PROGRAM PRG_MotorDrive
VAR
	fbEnableAxes: FB_EnableAxes;
	fbHalt1: MC_Halt;
	fbMoveVelocityFw: MC_MoveVelocity;
	fbMoveVelocityBw: MC_MoveVelocity;
	fbTON1: TON;
	fbRTrigMoveFw: R_TRIG;
	fbRTrigMoveBw: R_TRIG;
	fbRTrigHalt: R_TRIG;
	nAutoState: INT;
	nSpeed: INT := 400; //degrees/sec
END_VAR

fbEnableAxes.bEnableAxes := TRUE;
fbRTrigMoveFW(CLK:=GVL.bButtonFw, Q=>);
fbRTrigMoveBW(CLK:=GVL.bButtonBw, Q=>);
fbRTrigHalt(CLK:=GVL.bButtonHalt, Q=>);

IF fbRTrigMoveFw.Q THEN
	fbHalt1.Execute := FALSE;
	fbMoveVelocityBw.Execute := FALSE;
	fbMoveVelocityFw.Execute := TRUE;
END_IF

IF fbRTrigMoveBw.Q THEN
	fbHalt1.Execute := FALSE;
	fbMoveVelocityFw.Execute := FALSE;
	fbMoveVelocityBw.Execute := TRUE;
END_IF

IF fbRTrigHalt.Q THEN
	fbHalt1.Execute := TRUE;
	fbMoveVelocityFw.Execute := FALSE;
	fbMoveVelocityBw.Execute := FALSE;
END_IF

IF GVL.bButtonAuto THEN
	CASE nAutoState OF
		0: //Initialize auto motion
			fbHalt1.Execute := FALSE;
			fbMoveVelocityFw.Execute := FALSE;
			fbMoveVelocityBw.Execute := FALSE;
			nAutoState := 1;
		1: //Move forward
			fbTON1(IN:=TRUE, PT:=T#4S, Q=>, ET=>);
			fbMoveVelocityFw.Execute := TRUE;
			IF fbTON1.Q THEN
				fbTON1(IN:=FALSE);
				nAutoState := 2;	
			END_IF
		2: //Halt
			fbTON1(IN:=TRUE, PT:=T#2S, Q=>, ET=>);
			fbMoveVelocityFw.Execute := FALSE;
			fbHalt1.Execute := TRUE;
			IF fbTON1.Q THEN
				fbTON1(IN:=FALSE);
				nAutoState := 3;	
			END_IF
		3: //Move backward
			fbTON1(IN:=TRUE, PT:=T#4S, Q=>, ET=>);
			fbHalt1.Execute := FALSE;
			fbMoveVelocityBw.Execute := TRUE;
			IF fbTON1.Q THEN
				fbTON1(IN:=FALSE);
				nAutoState := 4;	
			END_IF
		4: //Halt again
			fbTON1(IN:=TRUE, PT:=T#2S, Q=>, ET=>);
			fbMoveVelocityBw.Execute := FALSE;
			fbHalt1.Execute := TRUE;
			IF fbTON1.Q THEN
				fbTON1(IN:=FALSE);
				nAutoState := 0;	
			END_IF
	END_CASE
END_IF

A_EnableAxes();
A_MoveVelocityFw();
A_MoveVelocityBw();
A_Halt();

ACTION A_EnableAxes:
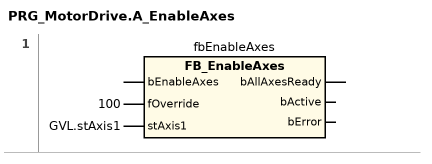
// NETWORK 1
fbEnableAxes(fOverride := 100, stAxis1 := GVL.stAxis1); // FB_EnableAxes
END_ACTION

ACTION A_Halt:
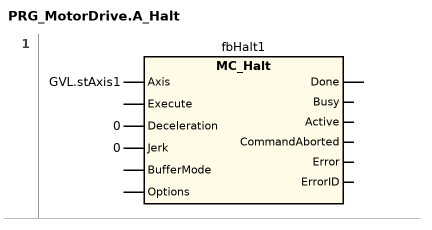
// NETWORK 1
fbHalt1(Axis := GVL.stAxis1, Deceleration := 0, Jerk := 0); // MC_Halt
END_ACTION

ACTION A_MoveVelocityBw:
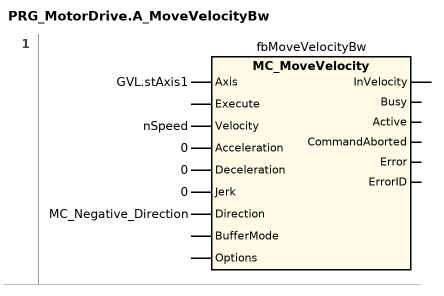
// NETWORK 1
fbMoveVelocityBw(
    Axis := GVL.stAxis1,
    Velocity := nSpeed,
    Acceleration := 0,
    Deceleration := 0,
    Jerk := 0,
    Direction := MC_Negative_Direction); // MC_MoveVelocity
END_ACTION

ACTION A_MoveVelocityFw:
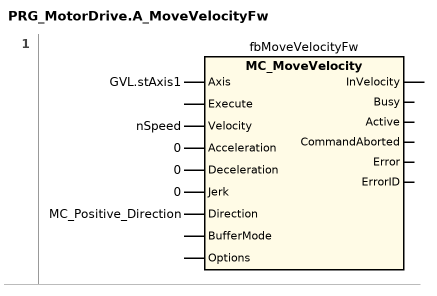
// NETWORK 1
fbMoveVelocityFw(
    Axis := GVL.stAxis1,
    Velocity := nSpeed,
    Acceleration := 0,
    Deceleration := 0,
    Jerk := 0,
    Direction := MC_Positive_Direction); // MC_MoveVelocity
END_ACTION

END_PROGRAM

(* stored: Version 1.1.0.1, ProductVersion 3.1.4024.12
   POU PRG_MotorDrive: Id {ad80292d-9aa9-4c68-b2fb-41bd24e30074}, SpecialFunc None
   Action A_EnableAxes: Id {4df17dcf-40b0-4a4e-9155-e0012275349a}
   Action A_Halt: Id {ac61f037-26e5-4c8a-a21e-6dbedfe6e82a}
   Action A_MoveVelocityBw: Id {92c62f3d-0340-48ba-8853-49b202b4035f}
   Action A_MoveVelocityFw: Id {81a3e208-9c92-49fe-bf3a-17f4b11c4149} *)
